// Mitsubishi GX Works2 project: 모터실린더연습   PLC: Q02/Q02H

PROGRAM MAIN
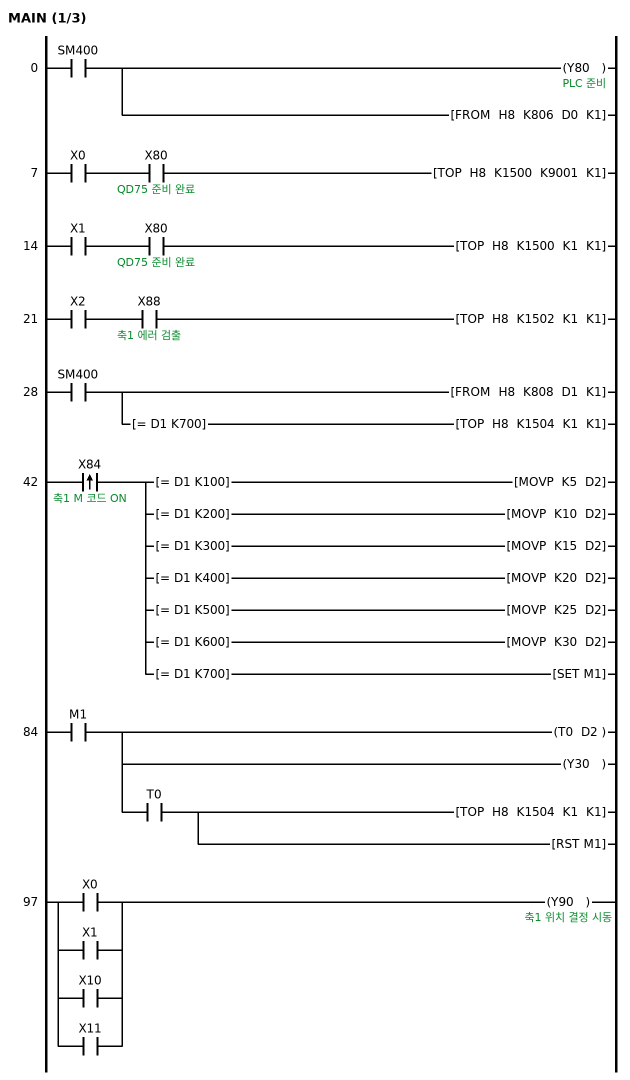
0     LD      SM400
      OUT     Y80  ; PLC 준비
      FROM    H8 K806 D0 K1
7     LD      X0
      AND     X80  ; QD75 준비 완료
      TOP     H8 K1500 K9001 K1
14    LD      X1
      AND     X80  ; QD75 준비 완료
      TOP     H8 K1500 K1 K1
21    LD      X2
      AND     X88  ; 축1 에러 검출
      TOP     H8 K1502 K1 K1
28    LD      SM400
      FROM    H8 K808 D1 K1
      AND=    D1 K700
      TOP     H8 K1504 K1 K1
42    LDP     X84  ; 축1 M 코드 ON
      MPS
      AND=    D1 K100
      MOVP    K5 D2
      MRD
      AND=    D1 K200
      MOVP    K10 D2
      MRD
      AND=    D1 K300
      MOVP    K15 D2
      MRD
      AND=    D1 K400
      MOVP    K20 D2
      MRD
      AND=    D1 K500
      MOVP    K25 D2
      MRD
      AND=    D1 K600
      MOVP    K30 D2
      MPP
      AND=    D1 K700
      SET     M1
84    LD      M1
      OUT     T0 D2
      OUT     Y30
      AND     T0
      TOP     H8 K1504 K1 K1
      RST     M1
97    LD      X0
      OR      X1
      OR      X10
      OR      X11
      OUT     Y90  ; 축1 위치 결정 시동
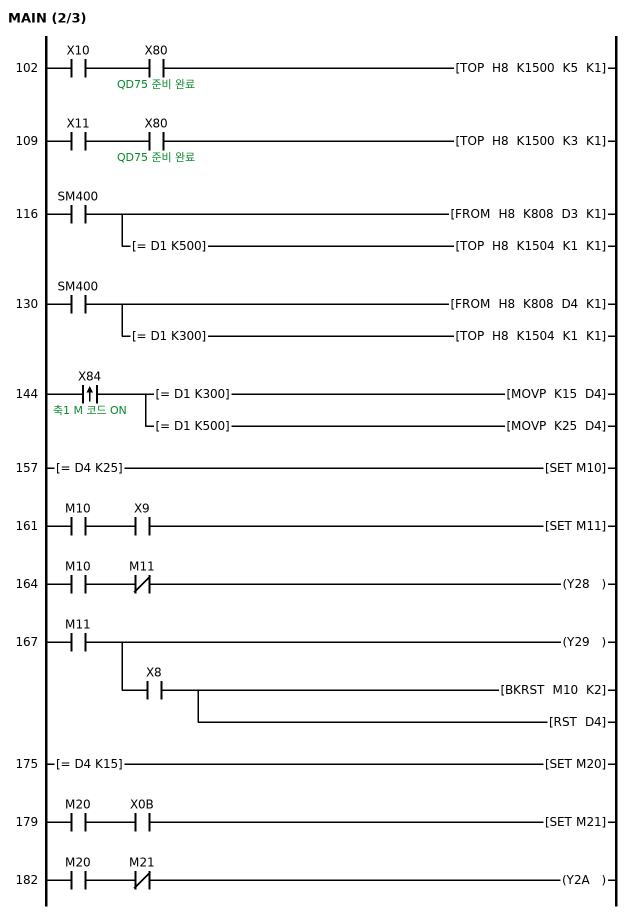
102   LD      X10
      AND     X80  ; QD75 준비 완료
      TOP     H8 K1500 K5 K1
109   LD      X11
      AND     X80  ; QD75 준비 완료
      TOP     H8 K1500 K3 K1
116   LD      SM400
      FROM    H8 K808 D3 K1
      AND=    D1 K500
      TOP     H8 K1504 K1 K1
130   LD      SM400
      FROM    H8 K808 D4 K1
      AND=    D1 K300
      TOP     H8 K1504 K1 K1
144   LDP     X84  ; 축1 M 코드 ON
      MPS
      AND=    D1 K300
      MOVP    K15 D4
      MPP
      AND=    D1 K500
      MOVP    K25 D4
157   LD=     D4 K25
      SET     M10
161   LD      M10
      AND     X9
      SET     M11
164   LD      M10
      ANI     M11
      OUT     Y28
167   LD      M11
      OUT     Y29
      AND     X8
      BKRST   M10 K2
      RST     D4
175   LD=     D4 K15
      SET     M20
179   LD      M20
      AND     X0B
      SET     M21
182   LD      M20
      ANI     M21
      OUT     Y2A
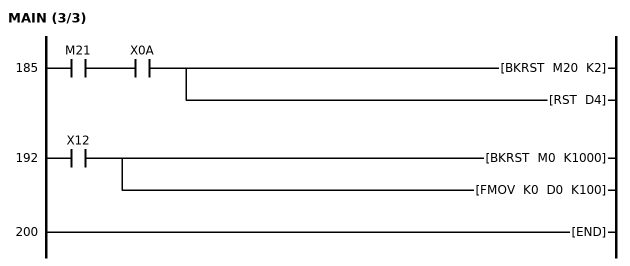
185   LD      M21
      AND     X0A
      BKRST   M20 K2
      RST     D4
192   LD      X12
      BKRST   M0 K1000
      FMOV    K0 D0 K100
200   END
END_PROGRAM

// device comments not shown above
X81  ; 동기용 플래그
X85  ; 축2 M 코드 ON
X89  ; 축2 에러 검출
X8C  ; 축1 BUSY
X8D  ; 축2 BUSY
X90  ; 축1 시동 완료
X91  ; 축2 시동 완료
X94  ; 축1 위치 결정 완료
X95  ; 축2 위치 결정 완료
Y84  ; 축1 축 정지
Y85  ; 축2 축 정지
Y88  ; 축1 정운전 JOG 시동
Y89  ; 축1 역운전 JOG 시동
Y8A  ; 축2 정운전 JOG 시동
Y8B  ; 축2 역운전 JOG 시동
Y91  ; 축2 위치 결정 시동
Y94  ; 축1 실행 금지 플래그
Y95  ; 축2 실행 금지 플래그
